// ---- DUTs/IO/Boxes/AT2042_33A3DF1B.TcDUT
{attribute 'GeneratedUsingTerminal: AT2042-5250-0019'}
{attribute addProperty BoxType "AT2042-5250-0019"}
{attribute addProperty Description "AT2042-5250 Sensor line with feed (B23-Connector), +45°"}
{attribute addProperty Physics "K"}
{attribute addProperty Id "FB_InputsAT %I*FB_Inputs_4BC4AA0166FB_OutputsAT %Q*FB_Outputs_DAFD38E02WcStateAT %I*WcState_9091E0EB2InfoDataAT %I*InfoData_A7436BC610"}
{attribute addProperty CRC "866377499"}
{attribute addProperty Size "80"}
TYPE AT2042_33A3DF1B EXTENDS EtcSlaveTerminalBase_947E5A46 :
STRUCT
	{attribute addProperty Name "FB_Inputs"}
	FB_Inputs : FB_Inputs_4BC4AA01;
	{attribute addProperty Name "FB_Outputs"}
	FB_Outputs : FB_Outputs_DAFD38E0;
	{attribute addProperty Name "WcState"}
	WcState : WcState_9091E0EB;
	{attribute addProperty Name "InfoData"}
	InfoData : InfoData_A7436BC6;
END_STRUCT
END_TYPE

// ---- DUTs/IO/Boxes/AT2041_33A3DF1B.TcDUT
{attribute 'GeneratedUsingTerminal: AT2041-5250-0019'}
{attribute addProperty BoxType "AT2041-5250-0019"}
{attribute addProperty Description "AT2041-5250 Sensor line with feed, +45°"}
{attribute addProperty Physics "K"}
{attribute addProperty Id "FB_InputsAT %I*FB_Inputs_4BC4AA0166FB_OutputsAT %Q*FB_Outputs_DAFD38E02WcStateAT %I*WcState_9091E0EB2InfoDataAT %I*InfoData_A7436BC610"}
{attribute addProperty CRC "866377499"}
{attribute addProperty Size "80"}
TYPE AT2041_33A3DF1B EXTENDS EtcSlaveTerminalBase_947E5A46 :
STRUCT
	{attribute addProperty Name "FB_Inputs"}
	FB_Inputs : FB_Inputs_4BC4AA01;
	{attribute addProperty Name "FB_Outputs"}
	FB_Outputs : FB_Outputs_DAFD38E0;
	{attribute addProperty Name "WcState"}
	WcState : WcState_9091E0EB;
	{attribute addProperty Name "InfoData"}
	InfoData : InfoData_A7436BC6;
END_STRUCT
END_TYPE

// ---- DUTs/IO/Boxes/AT2040_33A3DF1B.TcDUT
{attribute 'GeneratedUsingTerminal: AT2040-5250-0019'}
{attribute addProperty BoxType "AT2040-5250-0019"}
{attribute addProperty Description "AT2040-5250 Sensor line +45°"}
{attribute addProperty Physics "K"}
{attribute addProperty Id "FB_InputsAT %I*FB_Inputs_4BC4AA0166FB_OutputsAT %Q*FB_Outputs_DAFD38E02WcStateAT %I*WcState_9091E0EB2InfoDataAT %I*InfoData_A7436BC610"}
{attribute addProperty CRC "866377499"}
{attribute addProperty Size "80"}
TYPE AT2040_33A3DF1B EXTENDS EtcSlaveTerminalBase_947E5A46 :
STRUCT
	{attribute addProperty Name "FB_Inputs"}
	FB_Inputs : FB_Inputs_4BC4AA01;
	{attribute addProperty Name "FB_Outputs"}
	FB_Outputs : FB_Outputs_DAFD38E0;
	{attribute addProperty Name "WcState"}
	WcState : WcState_9091E0EB;
	{attribute addProperty Name "InfoData"}
	InfoData : InfoData_A7436BC6;
END_STRUCT
END_TYPE

// ---- DUTs/IO/Boxes/AT2042_2EA6C9BF.TcDUT
{attribute 'GeneratedUsingTerminal: AT2042-0250-0024'}
{attribute addProperty BoxType "AT2042-0250-0024"}
{attribute addProperty Description "AT2042-0250 Motor module with feed (B23-Connector), +45°, 250 mm, 48V"}
{attribute addProperty Physics "YKY"}
{attribute addProperty Id "CC_InputsAT %I*CC_Inputs_2C1C9EE032CC_OutputsAT %Q*CC_Outputs_69F9BE1432WcStateAT %I*WcState_9091E0EB2InfoDataAT %I*InfoData_BEF6B88E18"}
{attribute addProperty CRC "782682559"}
{attribute addProperty Size "84"}
TYPE AT2042_2EA6C9BF EXTENDS EtcSlaveBoxBase_77A0E4A7 :
STRUCT
	{attribute addProperty Name "CC_Inputs"}
	CC_Inputs : CC_Inputs_2C1C9EE0;
	{attribute addProperty Name "CC_Outputs"}
	CC_Outputs : CC_Outputs_69F9BE14;
	{attribute addProperty Name "WcState"}
	WcState : WcState_9091E0EB;
	{attribute addProperty Name "InfoData"}
	InfoData : InfoData_BEF6B88E;
END_STRUCT
END_TYPE

// ---- DUTs/IO/Boxes/AT2025_33A3DF1B.TcDUT
{attribute 'GeneratedUsingTerminal: AT2025-5250-0019'}
{attribute addProperty BoxType "AT2025-5250-0019"}
{attribute addProperty Description "AT2025-5250 Sensor line -22.5°"}
{attribute addProperty Physics "K"}
{attribute addProperty Id "FB_InputsAT %I*FB_Inputs_4BC4AA0166FB_OutputsAT %Q*FB_Outputs_DAFD38E02WcStateAT %I*WcState_9091E0EB2InfoDataAT %I*InfoData_A7436BC610"}
{attribute addProperty CRC "866377499"}
{attribute addProperty Size "80"}
TYPE AT2025_33A3DF1B EXTENDS EtcSlaveTerminalBase_947E5A46 :
STRUCT
	{attribute addProperty Name "FB_Inputs"}
	FB_Inputs : FB_Inputs_4BC4AA01;
	{attribute addProperty Name "FB_Outputs"}
	FB_Outputs : FB_Outputs_DAFD38E0;
	{attribute addProperty Name "WcState"}
	WcState : WcState_9091E0EB;
	{attribute addProperty Name "InfoData"}
	InfoData : InfoData_A7436BC6;
END_STRUCT
END_TYPE

// ---- DUTs/IO/Boxes/AT2050_2EA6C9BF.TcDUT
{attribute 'GeneratedUsingTerminal: AT2050-0500-0016'}
{attribute addProperty BoxType "AT2050-0500-0016"}
{attribute addProperty Description "AT2050-0500 Motor module, 90° clothoid, EtherCAT In, 50V"}
{attribute addProperty Physics "YKY"}
{attribute addProperty Id "CC_InputsAT %I*CC_Inputs_2C1C9EE032CC_OutputsAT %Q*CC_Outputs_69F9BE1432WcStateAT %I*WcState_9091E0EB2InfoDataAT %I*InfoData_BEF6B88E18"}
{attribute addProperty CRC "782682559"}
{attribute addProperty Size "84"}
TYPE AT2050_2EA6C9BF EXTENDS EtcSlaveBoxBase_77A0E4A7 :
STRUCT
	{attribute addProperty Name "CC_Inputs"}
	CC_Inputs : CC_Inputs_2C1C9EE0;
	{attribute addProperty Name "CC_Outputs"}
	CC_Outputs : CC_Outputs_69F9BE14;
	{attribute addProperty Name "WcState"}
	WcState : WcState_9091E0EB;
	{attribute addProperty Name "InfoData"}
	InfoData : InfoData_BEF6B88E;
END_STRUCT
END_TYPE

// ---- DUTs/IO/Boxes/AT2021_33A3DF1B.TcDUT
{attribute 'GeneratedUsingTerminal: AT2021-5250-0019'}
{attribute addProperty BoxType "AT2021-5250-0019"}
{attribute addProperty Description "AT2021-5250 Sensor line with feed, +22.5°"}
{attribute addProperty Physics "K"}
{attribute addProperty Id "FB_InputsAT %I*FB_Inputs_4BC4AA0166FB_OutputsAT %Q*FB_Outputs_DAFD38E02WcStateAT %I*WcState_9091E0EB2InfoDataAT %I*InfoData_A7436BC610"}
{attribute addProperty CRC "866377499"}
{attribute addProperty Size "80"}
TYPE AT2021_33A3DF1B EXTENDS EtcSlaveTerminalBase_947E5A46 :
STRUCT
	{attribute addProperty Name "FB_Inputs"}
	FB_Inputs : FB_Inputs_4BC4AA01;
	{attribute addProperty Name "FB_Outputs"}
	FB_Outputs : FB_Outputs_DAFD38E0;
	{attribute addProperty Name "WcState"}
	WcState : WcState_9091E0EB;
	{attribute addProperty Name "InfoData"}
	InfoData : InfoData_A7436BC6;
END_STRUCT
END_TYPE

// ---- DUTs/IO/Boxes/AT2020_33A3DF1B.TcDUT
{attribute 'GeneratedUsingTerminal: AT2020-5250-0019'}
{attribute addProperty BoxType "AT2020-5250-0019"}
{attribute addProperty Description "AT2020-5250 Sensor line +22.5°"}
{attribute addProperty Physics "K"}
{attribute addProperty Id "FB_InputsAT %I*FB_Inputs_4BC4AA0166FB_OutputsAT %Q*FB_Outputs_DAFD38E02WcStateAT %I*WcState_9091E0EB2InfoDataAT %I*InfoData_A7436BC610"}
{attribute addProperty CRC "866377499"}
{attribute addProperty Size "80"}
TYPE AT2020_33A3DF1B EXTENDS EtcSlaveTerminalBase_947E5A46 :
STRUCT
	{attribute addProperty Name "FB_Inputs"}
	FB_Inputs : FB_Inputs_4BC4AA01;
	{attribute addProperty Name "FB_Outputs"}
	FB_Outputs : FB_Outputs_DAFD38E0;
	{attribute addProperty Name "WcState"}
	WcState : WcState_9091E0EB;
	{attribute addProperty Name "InfoData"}
	InfoData : InfoData_A7436BC6;
END_STRUCT
END_TYPE

// ---- DUTs/IO/Boxes/AT2001_33A3DF1B.TcDUT
{attribute 'GeneratedUsingTerminal: AT2001-5250-0017'}
{attribute addProperty BoxType "AT2001-5250-0017"}
{attribute addProperty Description "AT2001-5250 Sensor line with feed"}
{attribute addProperty Physics "K"}
{attribute addProperty Id "FB_InputsAT %I*FB_Inputs_4BC4AA0166FB_OutputsAT %Q*FB_Outputs_DAFD38E02WcStateAT %I*WcState_9091E0EB2InfoDataAT %I*InfoData_A7436BC610"}
{attribute addProperty CRC "866377499"}
{attribute addProperty Size "80"}
TYPE AT2001_33A3DF1B EXTENDS EtcSlaveTerminalBase_947E5A46 :
STRUCT
	{attribute addProperty Name "FB_Inputs"}
	FB_Inputs : FB_Inputs_4BC4AA01;
	{attribute addProperty Name "FB_Outputs"}
	FB_Outputs : FB_Outputs_DAFD38E0;
	{attribute addProperty Name "WcState"}
	WcState : WcState_9091E0EB;
	{attribute addProperty Name "InfoData"}
	InfoData : InfoData_A7436BC6;
END_STRUCT
END_TYPE

// ---- DUTs/IO/Boxes/AT2002_33A3DF1B.TcDUT
{attribute 'GeneratedUsingTerminal: AT2002-5249-0018'}
{attribute addProperty BoxType "AT2002-5249-0018"}
{attribute addProperty Description "AT2002-5249 Sensor line (Track management) with feed"}
{attribute addProperty Physics "K"}
{attribute addProperty Id "FB_InputsAT %I*FB_Inputs_4BC4AA0166FB_OutputsAT %Q*FB_Outputs_DAFD38E02WcStateAT %I*WcState_9091E0EB2InfoDataAT %I*InfoData_A7436BC610"}
{attribute addProperty CRC "866377499"}
{attribute addProperty Size "80"}
TYPE AT2002_33A3DF1B EXTENDS EtcSlaveTerminalBase_947E5A46 :
STRUCT
	{attribute addProperty Name "FB_Inputs"}
	FB_Inputs : FB_Inputs_4BC4AA01;
	{attribute addProperty Name "FB_Outputs"}
	FB_Outputs : FB_Outputs_DAFD38E0;
	{attribute addProperty Name "WcState"}
	WcState : WcState_9091E0EB;
	{attribute addProperty Name "InfoData"}
	InfoData : InfoData_A7436BC6;
END_STRUCT
END_TYPE

// ---- DUTs/IO/Boxes/ATH2000_2EA6C9BF.TcDUT
{attribute 'GeneratedUsingTerminal: ATH2000-0250-0022'}
{attribute addProperty BoxType "ATH2000-0250-0022"}
{attribute addProperty Description "ATH2000-0250 Hygienic Motor module 250 mm, 48V"}
{attribute addProperty Physics "YKY"}
{attribute addProperty Id "CC_InputsAT %I*CC_Inputs_2C1C9EE032CC_OutputsAT %Q*CC_Outputs_69F9BE1432WcStateAT %I*WcState_9091E0EB2InfoDataAT %I*InfoData_BEF6B88E18"}
{attribute addProperty CRC "782682559"}
{attribute addProperty Size "84"}
TYPE ATH2000_2EA6C9BF EXTENDS EtcSlaveBoxBase_77A0E4A7 :
STRUCT
	{attribute addProperty Name "CC_Inputs"}
	CC_Inputs : CC_Inputs_2C1C9EE0;
	{attribute addProperty Name "CC_Outputs"}
	CC_Outputs : CC_Outputs_69F9BE14;
	{attribute addProperty Name "WcState"}
	WcState : WcState_9091E0EB;
	{attribute addProperty Name "InfoData"}
	InfoData : InfoData_BEF6B88E;
END_STRUCT
END_TYPE

// ---- DUTs/IO/Boxes/ATH2050_6EC099B7.TcDUT
{attribute 'GeneratedUsingTerminal: ATH2050-5501-0022'}
{attribute addProperty BoxType "ATH2050-5501-0022"}
{attribute addProperty Description "ATH2050-5501 Hygienic Sensor 90° clothoid, EtherCAT Out"}
{attribute addProperty Physics "K"}
{attribute addProperty Id "FB_InputsAT %I*FB_Inputs_391456510FB_OutputsAT %Q*FB_Outputs_DAFD38E02WcStateAT %I*WcState_9091E0EB2InfoDataAT %I*InfoData_A7436BC610"}
{attribute addProperty CRC "1858116023"}
{attribute addProperty Size "14"}
TYPE ATH2050_6EC099B7 EXTENDS EtcSlaveTerminalBase_947E5A46 :
STRUCT
	{attribute addProperty Name "FB_Inputs"}
	FB_Inputs : FB_Inputs_39145651;
	{attribute addProperty Name "FB_Outputs"}
	FB_Outputs : FB_Outputs_DAFD38E0;
	{attribute addProperty Name "WcState"}
	WcState : WcState_9091E0EB;
	{attribute addProperty Name "InfoData"}
	InfoData : InfoData_A7436BC6;
END_STRUCT
END_TYPE

// ---- DUTs/IO/Boxes/ATH2040_41437DDC.TcDUT
{attribute 'GeneratedUsingTerminal: ATH2040-5250-0022'}
{attribute addProperty BoxType "ATH2040-5250-0022"}
{attribute addProperty Description "ATH2040-5250 Hygienic Sensor +45°"}
{attribute addProperty Physics "K"}
{attribute addProperty Id "FB_InputsAT %I*FB_Inputs_01C600450FB_OutputsAT %Q*FB_Outputs_DAFD38E02WcStateAT %I*WcState_9091E0EB2InfoDataAT %I*InfoData_A7436BC610"}
{attribute addProperty CRC "1094942172"}
{attribute addProperty Size "14"}
TYPE ATH2040_41437DDC EXTENDS EtcSlaveTerminalBase_947E5A46 :
STRUCT
	{attribute addProperty Name "FB_Inputs"}
	FB_Inputs : FB_Inputs_01C60045;
	{attribute addProperty Name "FB_Outputs"}
	FB_Outputs : FB_Outputs_DAFD38E0;
	{attribute addProperty Name "WcState"}
	WcState : WcState_9091E0EB;
	{attribute addProperty Name "InfoData"}
	InfoData : InfoData_A7436BC6;
END_STRUCT
END_TYPE

// ---- DUTs/IO/Boxes/ATH2040_2EA6C9BF.TcDUT
{attribute 'GeneratedUsingTerminal: ATH2040-0250-0022'}
{attribute addProperty BoxType "ATH2040-0250-0022"}
{attribute addProperty Description "ATH2040-0250 Hygienic Motor module +45°, 250mm, 48V"}
{attribute addProperty Physics "YKY"}
{attribute addProperty Id "CC_InputsAT %I*CC_Inputs_2C1C9EE032CC_OutputsAT %Q*CC_Outputs_69F9BE1432WcStateAT %I*WcState_9091E0EB2InfoDataAT %I*InfoData_BEF6B88E18"}
{attribute addProperty CRC "782682559"}
{attribute addProperty Size "84"}
TYPE ATH2040_2EA6C9BF EXTENDS EtcSlaveBoxBase_77A0E4A7 :
STRUCT
	{attribute addProperty Name "CC_Inputs"}
	CC_Inputs : CC_Inputs_2C1C9EE0;
	{attribute addProperty Name "CC_Outputs"}
	CC_Outputs : CC_Outputs_69F9BE14;
	{attribute addProperty Name "WcState"}
	WcState : WcState_9091E0EB;
	{attribute addProperty Name "InfoData"}
	InfoData : InfoData_BEF6B88E;
END_STRUCT
END_TYPE

// ---- DUTs/IO/Boxes/ATH2050_2EA6C9BF.TcDUT
{attribute 'GeneratedUsingTerminal: ATH2050-0500-0022'}
{attribute addProperty BoxType "ATH2050-0500-0022"}
{attribute addProperty Description "ATH2050-0500 Hygienic Motor module 90° clothoid, EtherCAT In"}
{attribute addProperty Physics "YKY"}
{attribute addProperty Id "CC_InputsAT %I*CC_Inputs_2C1C9EE032CC_OutputsAT %Q*CC_Outputs_69F9BE1432WcStateAT %I*WcState_9091E0EB2InfoDataAT %I*InfoData_BEF6B88E18"}
{attribute addProperty CRC "782682559"}
{attribute addProperty Size "84"}
TYPE ATH2050_2EA6C9BF EXTENDS EtcSlaveBoxBase_77A0E4A7 :
STRUCT
	{attribute addProperty Name "CC_Inputs"}
	CC_Inputs : CC_Inputs_2C1C9EE0;
	{attribute addProperty Name "CC_Outputs"}
	CC_Outputs : CC_Outputs_69F9BE14;
	{attribute addProperty Name "WcState"}
	WcState : WcState_9091E0EB;
	{attribute addProperty Name "InfoData"}
	InfoData : InfoData_BEF6B88E;
END_STRUCT
END_TYPE

// ---- DUTs/IO/Boxes/ATH2000_D874080E.TcDUT
{attribute 'GeneratedUsingTerminal: ATH2000-5250-0022'}
{attribute addProperty BoxType "ATH2000-5250-0022"}
{attribute addProperty Description "ATH2000-5250 Hygienic Sensor line"}
{attribute addProperty Physics "K"}
{attribute addProperty Id "FB_InputsAT %I*FB_Inputs_2D6658510FB_OutputsAT %Q*FB_Outputs_DAFD38E02WcStateAT %I*WcState_9091E0EB2InfoDataAT %I*InfoData_A7436BC610"}
{attribute addProperty CRC "3631482894"}
{attribute addProperty Size "14"}
TYPE ATH2000_D874080E EXTENDS EtcSlaveTerminalBase_947E5A46 :
STRUCT
	{attribute addProperty Name "FB_Inputs"}
	FB_Inputs : FB_Inputs_2D665851;
	{attribute addProperty Name "FB_Outputs"}
	FB_Outputs : FB_Outputs_DAFD38E0;
	{attribute addProperty Name "WcState"}
	WcState : WcState_9091E0EB;
	{attribute addProperty Name "InfoData"}
	InfoData : InfoData_A7436BC6;
END_STRUCT
END_TYPE

// ---- DUTs/IO/Devices/SyncUnitTask_2D604ED5.TcDUT
{attribute 'GeneratedUsingTerminal: IODEVICETYPE_ETHERCATPROT'}
{attribute addProperty BoxType "IODEVICETYPE_ETHERCATPROT"}
{attribute addProperty Id "WcStateAT %I*WcState_0B2B16F91InfoDataAT %I*InfoData_2A97D6CF8"}
{attribute addProperty CRC "761286357"}
{attribute addProperty Size "9"}
TYPE SyncUnitTask_2D604ED5 :
STRUCT
	{attribute addProperty Name "WcState"}
	WcState : WcState_0B2B16F9;
	{attribute addProperty Name "InfoData"}
	InfoData : InfoData_2A97D6CF;
END_STRUCT
END_TYPE

// ---- DUTs/IO/Devices/SyncUnitTasks_6FEB8257.TcDUT
{attribute 'GeneratedUsingTerminal: '}
{attribute addProperty BoxType ""}
{attribute addProperty Id "unreferencedAT %I*SyncUnitTask_2D604ED59PlcTaskAT %I*SyncUnitTask_2D604ED59"}
{attribute addProperty CRC "1877705303"}
{attribute addProperty Size "18"}
TYPE SyncUnitTasks_6FEB8257 :
STRUCT
	{attribute addProperty Name "unreferenced"}
	unreferenced : SyncUnitTask_2D604ED5;
	{attribute addProperty Name "PlcTask"}
	PlcTask : SyncUnitTask_2D604ED5;
END_STRUCT
END_TYPE

// ---- DUTs/IO/Devices/SyncUnits_99E584AF.TcDUT
{attribute 'GeneratedUsingTerminal: '}
{attribute addProperty BoxType ""}
{attribute addProperty Id "_defaultAT %I*SyncUnitTasks_6FEB825718"}
{attribute addProperty CRC "2581955759"}
{attribute addProperty Size "18"}
TYPE SyncUnits_99E584AF :
STRUCT
	{attribute addProperty Name "_default"}
	_default : SyncUnitTasks_6FEB8257;
END_STRUCT
END_TYPE

// ---- DUTs/IO/Topology/A_0060_AT2020_0250_0019_AT2020_0250_29EE8276.TcDUT
{attribute 'GeneratedUsingTerminal: AT2020-0250-0019'}
{attribute addProperty BoxType "AT2020-0250-0019"}
{attribute addProperty Id "A_0085_AT2050_5500_0018_AT2050_5500AT2050_33A3DF1B80"}
{attribute addProperty CRC "703496822"}
{attribute addProperty Size "80"}
{attribute addProperty Name "A_0060(AT2020-0250-0019) (AT2020-0250)"}
TYPE A_0060_AT2020_0250_0019_AT2020_0250_29EE8276 EXTENDS AT2020_2EA6C9BF :
STRUCT
	{attribute addProperty Name "A_0085(AT2050-5500-0018) (AT2050-5500)"}
	{attribute addProperty PreviousPort "A_0060(AT2020-0250-0019) (AT2020-0250) : B"}
	A_0085_AT2050_5500_0018_AT2050_5500 : AT2050_33A3DF1B;
END_STRUCT
END_TYPE

// ---- DUTs/IO/Topology/A_0036_AT2040_0250_0021_0B822AE4.TcDUT
{attribute 'GeneratedUsingTerminal: AT2040-0250-0021'}
{attribute addProperty BoxType "AT2040-0250-0021"}
{attribute addProperty Id "A_0108_AT2000_5233_0019_AT2000_5233AT2000_33A3DF1B80"}
{attribute addProperty CRC "193080036"}
{attribute addProperty Size "80"}
{attribute addProperty Name "A_0036(AT2040-0250-0021)"}
TYPE A_0036_AT2040_0250_0021_0B822AE4 EXTENDS AT2040_2EA6C9BF :
STRUCT
	{attribute addProperty Name "A_0108(AT2000-5233-0019) (AT2000-5233)"}
	{attribute addProperty PreviousPort "A_0036(AT2040-0250-0021) : B"}
	A_0108_AT2000_5233_0019_AT2000_5233 : AT2000_33A3DF1B;
END_STRUCT
END_TYPE

// ---- DUTs/IO/Topology/A_0037_AT2040_0250_0022_033DCEC4.TcDUT
{attribute 'GeneratedUsingTerminal: AT2040-0250-0022'}
{attribute addProperty BoxType "AT2040-0250-0022"}
{attribute addProperty Id "A_0107_AT2000_5233_0018_AT2000_5233AT2000_33A3DF1B80"}
{attribute addProperty CRC "54382276"}
{attribute addProperty Size "80"}
{attribute addProperty Name "A_0037(AT2040-0250-0022)"}
TYPE A_0037_AT2040_0250_0022_033DCEC4 EXTENDS AT2040_2EA6C9BF :
STRUCT
	{attribute addProperty Name "A_0107(AT2000-5233-0018) (AT2000-5233)"}
	{attribute addProperty PreviousPort "A_0037(AT2040-0250-0022) : B"}
	A_0107_AT2000_5233_0018_AT2000_5233 : AT2000_33A3DF1B;
END_STRUCT
END_TYPE

// ---- DUTs/IO/Topology/A_0038_AT2040_0250_0023_C339CA0C.TcDUT
{attribute 'GeneratedUsingTerminal: AT2040-0250-0023'}
{attribute addProperty BoxType "AT2040-0250-0023"}
{attribute addProperty Id "A_0106_AT2026_5250_0019_AT2026_5250AT2026_33A3DF1B80"}
{attribute addProperty CRC "3275344396"}
{attribute addProperty Size "80"}
{attribute addProperty Name "A_0038(AT2040-0250-0023)"}
TYPE A_0038_AT2040_0250_0023_C339CA0C EXTENDS AT2040_2EA6C9BF :
STRUCT
	{attribute addProperty Name "A_0106(AT2026-5250-0019) (AT2026-5250)"}
	{attribute addProperty PreviousPort "A_0038(AT2040-0250-0023) : B"}
	A_0106_AT2026_5250_0019_AT2026_5250 : AT2026_33A3DF1B;
END_STRUCT
END_TYPE

// ---- DUTs/IO/Topology/A_0039_AT2040_0250_0024_375958EA.TcDUT
{attribute 'GeneratedUsingTerminal: AT2040-0250-0024'}
{attribute addProperty BoxType "AT2040-0250-0024"}
{attribute addProperty Id "A_0105_AT2026_5250_0018_AT2026_5250AT2026_33A3DF1B80"}
{attribute addProperty CRC "928602346"}
{attribute addProperty Size "80"}
{attribute addProperty Name "A_0039(AT2040-0250-0024)"}
TYPE A_0039_AT2040_0250_0024_375958EA EXTENDS AT2040_2EA6C9BF :
STRUCT
	{attribute addProperty Name "A_0105(AT2026-5250-0018) (AT2026-5250)"}
	{attribute addProperty PreviousPort "A_0039(AT2040-0250-0024) : B"}
	A_0105_AT2026_5250_0018_AT2026_5250 : AT2026_33A3DF1B;
END_STRUCT
END_TYPE

// ---- DUTs/IO/Topology/A_0040_AT2041_0250_0018_536500F2.TcDUT
{attribute 'GeneratedUsingTerminal: AT2041-0250-0018'}
{attribute addProperty BoxType "AT2041-0250-0018"}
{attribute addProperty Id "A_0104_AT2042_5250_0019_AT2042_5250AT2042_33A3DF1B80"}
{attribute addProperty CRC "1399128306"}
{attribute addProperty Size "80"}
{attribute addProperty Name "A_0040(AT2041-0250-0018)"}
TYPE A_0040_AT2041_0250_0018_536500F2 EXTENDS AT2041_2EA6C9BF :
STRUCT
	{attribute addProperty Name "A_0104(AT2042-5250-0019) (AT2042-5250)"}
	{attribute addProperty PreviousPort "A_0040(AT2041-0250-0018) : B"}
	A_0104_AT2042_5250_0019_AT2042_5250 : AT2042_33A3DF1B;
END_STRUCT
END_TYPE

// ---- DUTs/IO/Topology/A_0041_AT2041_0250_0019_F34F4056.TcDUT
{attribute 'GeneratedUsingTerminal: AT2041-0250-0019'}
{attribute addProperty BoxType "AT2041-0250-0019"}
{attribute addProperty Id "A_0103_AT2042_5250_0018_AT2042_5250AT2042_33A3DF1B80"}
{attribute addProperty CRC "4082057302"}
{attribute addProperty Size "80"}
{attribute addProperty Name "A_0041(AT2041-0250-0019)"}
TYPE A_0041_AT2041_0250_0019_F34F4056 EXTENDS AT2041_2EA6C9BF :
STRUCT
	{attribute addProperty Name "A_0103(AT2042-5250-0018) (AT2042-5250)"}
	{attribute addProperty PreviousPort "A_0041(AT2041-0250-0019) : B"}
	A_0103_AT2042_5250_0018_AT2042_5250 : AT2042_33A3DF1B;
END_STRUCT
END_TYPE

// ---- DUTs/IO/Topology/A_0042_AT2041_0250_0020_5E65A51E.TcDUT
{attribute 'GeneratedUsingTerminal: AT2041-0250-0020'}
{attribute addProperty BoxType "AT2041-0250-0020"}
{attribute addProperty Id "A_0102_AT2041_5250_0019_AT2041_5250AT2041_33A3DF1B80"}
{attribute addProperty CRC "1583719710"}
{attribute addProperty Size "80"}
{attribute addProperty Name "A_0042(AT2041-0250-0020)"}
TYPE A_0042_AT2041_0250_0020_5E65A51E EXTENDS AT2041_2EA6C9BF :
STRUCT
	{attribute addProperty Name "A_0102(AT2041-5250-0019) (AT2041-5250)"}
	{attribute addProperty PreviousPort "A_0042(AT2041-0250-0020) : B"}
	A_0102_AT2041_5250_0019_AT2041_5250 : AT2041_33A3DF1B;
END_STRUCT
END_TYPE

// ---- DUTs/IO/Topology/A_0043_AT2041_0250_0021_AA0537F8.TcDUT
{attribute 'GeneratedUsingTerminal: AT2041-0250-0021'}
{attribute addProperty BoxType "AT2041-0250-0021"}
{attribute addProperty Id "A_0101_AT2041_5250_0018_AT2041_5250AT2041_33A3DF1B80"}
{attribute addProperty CRC "2852468728"}
{attribute addProperty Size "80"}
{attribute addProperty Name "A_0043(AT2041-0250-0021)"}
TYPE A_0043_AT2041_0250_0021_AA0537F8 EXTENDS AT2041_2EA6C9BF :
STRUCT
	{attribute addProperty Name "A_0101(AT2041-5250-0018) (AT2041-5250)"}
	{attribute addProperty PreviousPort "A_0043(AT2041-0250-0021) : B"}
	A_0101_AT2041_5250_0018_AT2041_5250 : AT2041_33A3DF1B;
END_STRUCT
END_TYPE

// ---- DUTs/IO/Topology/A_0044_AT2041_0250_0022_5A9A39BA.TcDUT
{attribute 'GeneratedUsingTerminal: AT2041-0250-0022'}
{attribute addProperty BoxType "AT2041-0250-0022"}
{attribute addProperty Id "A_0100_AT2040_5250_0019_AT2040_5250AT2040_33A3DF1B80"}
{attribute addProperty CRC "1520056762"}
{attribute addProperty Size "80"}
{attribute addProperty Name "A_0044(AT2041-0250-0022)"}
TYPE A_0044_AT2041_0250_0022_5A9A39BA EXTENDS AT2041_2EA6C9BF :
STRUCT
	{attribute addProperty Name "A_0100(AT2040-5250-0019) (AT2040-5250)"}
	{attribute addProperty PreviousPort "A_0044(AT2041-0250-0022) : B"}
	A_0100_AT2040_5250_0019_AT2040_5250 : AT2040_33A3DF1B;
END_STRUCT
END_TYPE

// ---- DUTs/IO/Topology/A_0045_AT2041_0250_0023_51C662AC.TcDUT
{attribute 'GeneratedUsingTerminal: AT2041-0250-0023'}
{attribute addProperty BoxType "AT2041-0250-0023"}
{attribute addProperty Id "A_0099_AT2040_5250_0018_AT2040_5250AT2040_33A3DF1B80"}
{attribute addProperty CRC "1371955884"}
{attribute addProperty Size "80"}
{attribute addProperty Name "A_0045(AT2041-0250-0023)"}
TYPE A_0045_AT2041_0250_0023_51C662AC EXTENDS AT2041_2EA6C9BF :
STRUCT
	{attribute addProperty Name "A_0099(AT2040-5250-0018) (AT2040-5250)"}
	{attribute addProperty PreviousPort "A_0045(AT2041-0250-0023) : B"}
	A_0099_AT2040_5250_0018_AT2040_5250 : AT2040_33A3DF1B;
END_STRUCT
END_TYPE

// ---- DUTs/IO/Topology/A_0046_AT2042_0250_0024_1B20CF31.TcDUT
{attribute 'GeneratedUsingTerminal: AT2042-0250-0024'}
{attribute addProperty BoxType "AT2042-0250-0024"}
{attribute addProperty Id "A_0098_AT2025_5250_0019_AT2025_5250AT2025_33A3DF1B80"}
{attribute addProperty CRC "455135025"}
{attribute addProperty Size "80"}
{attribute addProperty Name "A_0046(AT2042-0250-0024)"}
TYPE A_0046_AT2042_0250_0024_1B20CF31 EXTENDS AT2042_2EA6C9BF :
STRUCT
	{attribute addProperty Name "A_0098(AT2025-5250-0019) (AT2025-5250)"}
	{attribute addProperty PreviousPort "A_0046(AT2042-0250-0024) : B"}
	A_0098_AT2025_5250_0019_AT2025_5250 : AT2025_33A3DF1B;
END_STRUCT
END_TYPE

// ---- DUTs/IO/Topology/A_0047_AT2050_0500_0016_139F2B11.TcDUT
{attribute 'GeneratedUsingTerminal: AT2050-0500-0016'}
{attribute addProperty BoxType "AT2050-0500-0016"}
{attribute addProperty Id "A_0097_AT2025_5250_0018_AT2025_5250AT2025_33A3DF1B80"}
{attribute addProperty CRC "329198353"}
{attribute addProperty Size "80"}
{attribute addProperty Name "A_0047(AT2050-0500-0016)"}
TYPE A_0047_AT2050_0500_0016_139F2B11 EXTENDS AT2050_2EA6C9BF :
STRUCT
	{attribute addProperty Name "A_0097(AT2025-5250-0018) (AT2025-5250)"}
	{attribute addProperty PreviousPort "A_0047(AT2050-0500-0016) : B"}
	A_0097_AT2025_5250_0018_AT2025_5250 : AT2025_33A3DF1B;
END_STRUCT
END_TYPE

// ---- DUTs/IO/Topology/A_0048_AT2050_0500_0017_3F977F47.TcDUT
{attribute 'GeneratedUsingTerminal: AT2050-0500-0017'}
{attribute addProperty BoxType "AT2050-0500-0017"}
{attribute addProperty Id "A_0096_AT2025_5250_0017_AT2025_5250AT2025_33A3DF1B80"}
{attribute addProperty CRC "1066893127"}
{attribute addProperty Size "80"}
{attribute addProperty Name "A_0048(AT2050-0500-0017)"}
TYPE A_0048_AT2050_0500_0017_3F977F47 EXTENDS AT2050_2EA6C9BF :
STRUCT
	{attribute addProperty Name "A_0096(AT2025-5250-0017) (AT2025-5250)"}
	{attribute addProperty PreviousPort "A_0048(AT2050-0500-0017) : B"}
	A_0096_AT2025_5250_0017_AT2025_5250 : AT2025_33A3DF1B;
END_STRUCT
END_TYPE

// ---- DUTs/IO/Topology/A_0049_AT2050_0500_0018_CBE655A8.TcDUT
{attribute 'GeneratedUsingTerminal: AT2050-0500-0018'}
{attribute addProperty BoxType "AT2050-0500-0018"}
{attribute addProperty Id "A_0095_AT2021_5250_0019_AT2021_5250AT2021_33A3DF1B80"}
{attribute addProperty CRC "3420870056"}
{attribute addProperty Size "80"}
{attribute addProperty Name "A_0049(AT2050-0500-0018)"}
TYPE A_0049_AT2050_0500_0018_CBE655A8 EXTENDS AT2050_2EA6C9BF :
STRUCT
	{attribute addProperty Name "A_0095(AT2021-5250-0019) (AT2021-5250)"}
	{attribute addProperty PreviousPort "A_0049(AT2050-0500-0018) : B"}
	A_0095_AT2021_5250_0019_AT2021_5250 : AT2021_33A3DF1B;
END_STRUCT
END_TYPE

// ---- DUTs/IO/Topology/A_0050_AT2050_0500_0019_15A3AE6F.TcDUT
{attribute 'GeneratedUsingTerminal: AT2050-0500-0019'}
{attribute addProperty BoxType "AT2050-0500-0019"}
{attribute addProperty Id "A_0094_AT2021_5250_0018_AT2021_5250AT2021_33A3DF1B80"}
{attribute addProperty CRC "363048559"}
{attribute addProperty Size "80"}
{attribute addProperty Name "A_0050(AT2050-0500-0019)"}
TYPE A_0050_AT2050_0500_0019_15A3AE6F EXTENDS AT2050_2EA6C9BF :
STRUCT
	{attribute addProperty Name "A_0094(AT2021-5250-0018) (AT2021-5250)"}
	{attribute addProperty PreviousPort "A_0050(AT2050-0500-0019) : B"}
	A_0094_AT2021_5250_0018_AT2021_5250 : AT2021_33A3DF1B;
END_STRUCT
END_TYPE

// ---- DUTs/IO/Topology/A_0051_AT2050_0500_0020_9B531B4E.TcDUT
{attribute 'GeneratedUsingTerminal: AT2050-0500-0020'}
{attribute addProperty BoxType "AT2050-0500-0020"}
{attribute addProperty Id "A_0093_AT2020_5250_0019_AT2020_5250AT2020_33A3DF1B80"}
{attribute addProperty CRC "2605914958"}
{attribute addProperty Size "80"}
{attribute addProperty Name "A_0051(AT2050-0500-0020)"}
TYPE A_0051_AT2050_0500_0020_9B531B4E EXTENDS AT2050_2EA6C9BF :
STRUCT
	{attribute addProperty Name "A_0093(AT2020-5250-0019) (AT2020-5250)"}
	{attribute addProperty PreviousPort "A_0051(AT2050-0500-0020) : B"}
	A_0093_AT2020_5250_0019_AT2020_5250 : AT2020_33A3DF1B;
END_STRUCT
END_TYPE

// ---- DUTs/IO/Topology/A_0052_AT2050_0500_0021_4516E089.TcDUT
{attribute 'GeneratedUsingTerminal: AT2050-0500-0021'}
{attribute addProperty BoxType "AT2050-0500-0021"}
{attribute addProperty Id "A_0092_AT2020_5250_0018_AT2020_5250AT2020_33A3DF1B80"}
{attribute addProperty CRC "1159127177"}
{attribute addProperty Size "80"}
{attribute addProperty Name "A_0052(AT2050-0500-0021)"}
TYPE A_0052_AT2050_0500_0021_4516E089 EXTENDS AT2050_2EA6C9BF :
STRUCT
	{attribute addProperty Name "A_0092(AT2020-5250-0018) (AT2020-5250)"}
	{attribute addProperty PreviousPort "A_0052(AT2050-0500-0021) : B"}
	A_0092_AT2020_5250_0018_AT2020_5250 : AT2020_33A3DF1B;
END_STRUCT
END_TYPE

// ---- DUTs/IO/Topology/A_0053_AT2050_0500_0022_433BDDFE.TcDUT
{attribute 'GeneratedUsingTerminal: AT2050-0500-0022'}
{attribute addProperty BoxType "AT2050-0500-0022"}
{attribute addProperty Id "A_0091_AT2020_5250_0017_AT2020_5250AT2020_33A3DF1B80"}
{attribute addProperty CRC "1127996926"}
{attribute addProperty Size "80"}
{attribute addProperty Name "A_0053(AT2050-0500-0022)"}
TYPE A_0053_AT2050_0500_0022_433BDDFE EXTENDS AT2050_2EA6C9BF :
STRUCT
	{attribute addProperty Name "A_0091(AT2020-5250-0017) (AT2020-5250)"}
	{attribute addProperty PreviousPort "A_0053(AT2050-0500-0022) : B"}
	A_0091_AT2020_5250_0017_AT2020_5250 : AT2020_33A3DF1B;
END_STRUCT
END_TYPE

// ---- DUTs/IO/Topology/A_0054_AT2050_0500_0023_B2F2DF55.TcDUT
{attribute 'GeneratedUsingTerminal: AT2050-0500-0023'}
{attribute addProperty BoxType "AT2050-0500-0023"}
{attribute addProperty Id "A_0090_AT2050_5501_0019_AT2050_5501AT2050_33A3DF1B80"}
{attribute addProperty CRC "3002261333"}
{attribute addProperty Size "80"}
{attribute addProperty Name "A_0054(AT2050-0500-0023)"}
TYPE A_0054_AT2050_0500_0023_B2F2DF55 EXTENDS AT2050_2EA6C9BF :
STRUCT
	{attribute addProperty Name "A_0090(AT2050-5501-0019) (AT2050-5501)"}
	{attribute addProperty PreviousPort "A_0054(AT2050-0500-0023) : B"}
	A_0090_AT2050_5501_0019_AT2050_5501 : AT2050_33A3DF1B;
END_STRUCT
END_TYPE

// ---- DUTs/IO/Topology/A_0055_AT2050_0500_0024_8D42A08D.TcDUT
{attribute 'GeneratedUsingTerminal: AT2050-0500-0024'}
{attribute addProperty BoxType "AT2050-0500-0024"}
{attribute addProperty Id "A_0089_AT2050_5501_0018_AT2050_5501AT2050_33A3DF1B80"}
{attribute addProperty CRC "2369953933"}
{attribute addProperty Size "80"}
{attribute addProperty Name "A_0055(AT2050-0500-0024)"}
TYPE A_0055_AT2050_0500_0024_8D42A08D EXTENDS AT2050_2EA6C9BF :
STRUCT
	{attribute addProperty Name "A_0089(AT2050-5501-0018) (AT2050-5501)"}
	{attribute addProperty PreviousPort "A_0055(AT2050-0500-0024) : B"}
	A_0089_AT2050_5501_0018_AT2050_5501 : AT2050_33A3DF1B;
END_STRUCT
END_TYPE

// ---- DUTs/IO/Topology/A_0056_AT2050_0501_0017_A14AF4DB.TcDUT
{attribute 'GeneratedUsingTerminal: AT2050-0501-0017'}
{attribute addProperty BoxType "AT2050-0501-0017"}
{attribute addProperty Id "A_0088_AT2050_5501_0017_AT2050_5501AT2050_33A3DF1B80"}
{attribute addProperty CRC "2706044123"}
{attribute addProperty Size "80"}
{attribute addProperty Name "A_0056(AT2050-0501-0017)"}
TYPE A_0056_AT2050_0501_0017_A14AF4DB EXTENDS AT2050_2EA6C9BF :
STRUCT
	{attribute addProperty Name "A_0088(AT2050-5501-0017) (AT2050-5501)"}
	{attribute addProperty PreviousPort "A_0056(AT2050-0501-0017) : B"}
	A_0088_AT2050_5501_0017_AT2050_5501 : AT2050_33A3DF1B;
END_STRUCT
END_TYPE

// ---- DUTs/IO/Topology/A_0057_AT2050_0501_0020_A9F510FB.TcDUT
{attribute 'GeneratedUsingTerminal: AT2050-0501-0020'}
{attribute addProperty BoxType "AT2050-0501-0020"}
{attribute addProperty Id "A_0087_AT2050_5501_0016_AT2050_5501AT2050_33A3DF1B80"}
{attribute addProperty CRC "2851410171"}
{attribute addProperty Size "80"}
{attribute addProperty Name "A_0057(AT2050-0501-0020)"}
TYPE A_0057_AT2050_0501_0020_A9F510FB EXTENDS AT2050_2EA6C9BF :
STRUCT
	{attribute addProperty Name "A_0087(AT2050-5501-0016) (AT2050-5501)"}
	{attribute addProperty PreviousPort "A_0057(AT2050-0501-0020) : B"}
	A_0087_AT2050_5501_0016_AT2050_5501 : AT2050_33A3DF1B;
END_STRUCT
END_TYPE

// ---- DUTs/IO/Topology/A_0058_AT2050_0501_0021_DD8E1090.TcDUT
{attribute 'GeneratedUsingTerminal: AT2050-0501-0021'}
{attribute addProperty BoxType "AT2050-0501-0021"}
{attribute addProperty Id "A_0086_AT2050_5500_0019_AT2050_5500AT2050_33A3DF1B80"}
{attribute addProperty CRC "3717075088"}
{attribute addProperty Size "80"}
{attribute addProperty Name "A_0058(AT2050-0501-0021)"}
TYPE A_0058_AT2050_0501_0021_DD8E1090 EXTENDS AT2050_2EA6C9BF :
STRUCT
	{attribute addProperty Name "A_0086(AT2050-5500-0019) (AT2050-5500)"}
	{attribute addProperty PreviousPort "A_0058(AT2050-0501-0021) : B"}
	A_0086_AT2050_5500_0019_AT2050_5500 : AT2050_33A3DF1B;
END_STRUCT
END_TYPE

// ---- DUTs/IO/Topology/A_0061_AT2020_0250_0023_AT2020_0250_2D9AB3DC.TcDUT
{attribute 'GeneratedUsingTerminal: AT2020-0250-0023'}
{attribute addProperty BoxType "AT2020-0250-0023"}
{attribute addProperty Id "A_0073_AT2000_5250_0016_AT2000_5250AT2000_33A3DF1B80"}
{attribute addProperty CRC "765113308"}
{attribute addProperty Size "80"}
{attribute addProperty Name "A_0061(AT2020-0250-0023) (AT2020-0250)"}
TYPE A_0061_AT2020_0250_0023_AT2020_0250_2D9AB3DC EXTENDS AT2020_2EA6C9BF :
STRUCT
	{attribute addProperty Name "A_0073(AT2000-5250-0016) (AT2000-5250)"}
	{attribute addProperty PreviousPort "A_0061(AT2020-0250-0023) (AT2020-0250) : B"}
	A_0073_AT2000_5250_0016_AT2000_5250 : AT2000_33A3DF1B;
END_STRUCT
END_TYPE

// ---- DUTs/IO/Topology/A_0062_AT2025_0250_0020_AT2025_0250_8DB0F378.TcDUT
{attribute 'GeneratedUsingTerminal: AT2025-0250-0020'}
{attribute addProperty BoxType "AT2025-0250-0020"}
{attribute addProperty Id "A_0074_AT2000_5250_0017_AT2000_5250AT2000_33A3DF1B80"}
{attribute addProperty CRC "2377184120"}
{attribute addProperty Size "80"}
{attribute addProperty Name "A_0062(AT2025-0250-0020) (AT2025-0250)"}
TYPE A_0062_AT2025_0250_0020_AT2025_0250_8DB0F378 EXTENDS AT2025_2EA6C9BF :
STRUCT
	{attribute addProperty Name "A_0074(AT2000-5250-0017) (AT2000-5250)"}
	{attribute addProperty PreviousPort "A_0062(AT2025-0250-0020) (AT2025-0250) : B"}
	A_0074_AT2000_5250_0017_AT2000_5250 : AT2000_33A3DF1B;
END_STRUCT
END_TYPE

// ---- DUTs/IO/Topology/A_0063_AT2025_0250_0022_AT2025_0250_E88F66A2.TcDUT
{attribute 'GeneratedUsingTerminal: AT2025-0250-0022'}
{attribute addProperty BoxType "AT2025-0250-0022"}
{attribute addProperty Id "A_0075_AT2000_5250_0019_AT2000_5250AT2000_33A3DF1B80"}
{attribute addProperty CRC "3901712034"}
{attribute addProperty Size "80"}
{attribute addProperty Name "A_0063(AT2025-0250-0022) (AT2025-0250)"}
TYPE A_0063_AT2025_0250_0022_AT2025_0250_E88F66A2 EXTENDS AT2025_2EA6C9BF :
STRUCT
	{attribute addProperty Name "A_0075(AT2000-5250-0019) (AT2000-5250)"}
	{attribute addProperty PreviousPort "A_0063(AT2025-0250-0022) (AT2025-0250) : B"}
	A_0075_AT2000_5250_0019_AT2000_5250 : AT2000_33A3DF1B;
END_STRUCT
END_TYPE

// ---- DUTs/IO/Topology/A_0064_AT2025_0250_0023_AT2025_0250_894F6FDC.TcDUT
{attribute 'GeneratedUsingTerminal: AT2025-0250-0023'}
{attribute addProperty BoxType "AT2025-0250-0023"}
{attribute addProperty Id "A_0076_AT2001_5250_0017_AT2001_5250AT2001_33A3DF1B80"}
{attribute addProperty CRC "2303684572"}
{attribute addProperty Size "80"}
{attribute addProperty Name "A_0064(AT2025-0250-0023) (AT2025-0250)"}
TYPE A_0064_AT2025_0250_0023_AT2025_0250_894F6FDC EXTENDS AT2025_2EA6C9BF :
STRUCT
	{attribute addProperty Name "A_0076(AT2001-5250-0017) (AT2001-5250)"}
	{attribute addProperty PreviousPort "A_0064(AT2025-0250-0023) (AT2025-0250) : B"}
	A_0076_AT2001_5250_0017_AT2001_5250 : AT2001_33A3DF1B;
END_STRUCT
END_TYPE

// ---- DUTs/IO/Topology/A_0065_AT2026_0250_0019_AT2026_0250_A5473B8A.TcDUT
{attribute 'GeneratedUsingTerminal: AT2026-0250-0019'}
{attribute addProperty BoxType "AT2026-0250-0019"}
{attribute addProperty Id "A_0077_AT2001_5250_0018_AT2001_5250AT2001_33A3DF1B80"}
{attribute addProperty CRC "2772908938"}
{attribute addProperty Size "80"}
{attribute addProperty Name "A_0065(AT2026-0250-0019) (AT2026-0250)"}
TYPE A_0065_AT2026_0250_0019_AT2026_0250_A5473B8A EXTENDS AT2026_2EA6C9BF :
STRUCT
	{attribute addProperty Name "A_0077(AT2001-5250-0018) (AT2001-5250)"}
	{attribute addProperty PreviousPort "A_0065(AT2026-0250-0019) (AT2026-0250) : B"}
	A_0077_AT2001_5250_0018_AT2001_5250 : AT2001_33A3DF1B;
END_STRUCT
END_TYPE

// ---- DUTs/IO/Topology/A_0066_AT2026_0250_0020_AT2026_0250_ADF8DFAA.TcDUT
{attribute 'GeneratedUsingTerminal: AT2026-0250-0020'}
{attribute addProperty BoxType "AT2026-0250-0020"}
{attribute addProperty Id "A_0078_AT2001_5250_0019_AT2001_5250AT2001_33A3DF1B80"}
{attribute addProperty CRC "2918768554"}
{attribute addProperty Size "80"}
{attribute addProperty Name "A_0066(AT2026-0250-0020) (AT2026-0250)"}
TYPE A_0066_AT2026_0250_0020_AT2026_0250_ADF8DFAA EXTENDS AT2026_2EA6C9BF :
STRUCT
	{attribute addProperty Name "A_0078(AT2001-5250-0019) (AT2001-5250)"}
	{attribute addProperty PreviousPort "A_0066(AT2026-0250-0020) (AT2026-0250) : B"}
	A_0078_AT2001_5250_0019_AT2001_5250 : AT2001_33A3DF1B;
END_STRUCT
END_TYPE

// ---- DUTs/IO/Topology/A_0067_AT2026_0250_0022_AT2026_0250_BF728FE6.TcDUT
{attribute 'GeneratedUsingTerminal: AT2026-0250-0022'}
{attribute addProperty BoxType "AT2026-0250-0022"}
{attribute addProperty Id "A_0079_AT2002_5249_0018_AT2002_5249AT2002_33A3DF1B80"}
{attribute addProperty CRC "3211956198"}
{attribute addProperty Size "80"}
{attribute addProperty Name "A_0067(AT2026-0250-0022) (AT2026-0250)"}
TYPE A_0067_AT2026_0250_0022_AT2026_0250_BF728FE6 EXTENDS AT2026_2EA6C9BF :
STRUCT
	{attribute addProperty Name "A_0079(AT2002-5249-0018) (AT2002-5249)"}
	{attribute addProperty PreviousPort "A_0067(AT2026-0250-0022) (AT2026-0250) : B"}
	A_0079_AT2002_5249_0018_AT2002_5249 : AT2002_33A3DF1B;
END_STRUCT
END_TYPE

// ---- DUTs/IO/Topology/A_0068_AT2026_0250_0024_AT2026_0250_71C01165.TcDUT
{attribute 'GeneratedUsingTerminal: AT2026-0250-0024'}
{attribute addProperty BoxType "AT2026-0250-0024"}
{attribute addProperty Id "A_0080_AT2002_5249_0019_AT2002_5249AT2002_33A3DF1B80"}
{attribute addProperty CRC "1908412773"}
{attribute addProperty Size "80"}
{attribute addProperty Name "A_0068(AT2026-0250-0024) (AT2026-0250)"}
TYPE A_0068_AT2026_0250_0024_AT2026_0250_71C01165 EXTENDS AT2026_2EA6C9BF :
STRUCT
	{attribute addProperty Name "A_0080(AT2002-5249-0019) (AT2002-5249)"}
	{attribute addProperty PreviousPort "A_0068(AT2026-0250-0024) (AT2026-0250) : B"}
	A_0080_AT2002_5249_0019_AT2002_5249 : AT2002_33A3DF1B;
END_STRUCT
END_TYPE

// ---- DUTs/IO/Topology/A_0069_AT2050_0501_0019_AT2050_0501_10255FA6.TcDUT
{attribute 'GeneratedUsingTerminal: AT2050-0501-0019'}
{attribute addProperty BoxType "AT2050-0501-0019"}
{attribute addProperty Id "A_0081_AT2002_5250_0018_AT2002_5250AT2002_33A3DF1B80"}
{attribute addProperty CRC "270884774"}
{attribute addProperty Size "80"}
{attribute addProperty Name "A_0069(AT2050-0501-0019) (AT2050-0501)"}
TYPE A_0069_AT2050_0501_0019_AT2050_0501_10255FA6 EXTENDS AT2050_2EA6C9BF :
STRUCT
	{attribute addProperty Name "A_0081(AT2002-5250-0018) (AT2002-5250)"}
	{attribute addProperty PreviousPort "A_0069(AT2050-0501-0019) (AT2050-0501) : B"}
	A_0081_AT2002_5250_0018_AT2002_5250 : AT2002_33A3DF1B;
END_STRUCT
END_TYPE

// ---- DUTs/IO/Topology/A_0070_AT2050_0501_0022_AT2050_0501_E445CD40.TcDUT
{attribute 'GeneratedUsingTerminal: AT2050-0501-0022'}
{attribute addProperty BoxType "AT2050-0501-0022"}
{attribute addProperty Id "A_0082_AT2002_5250_0019_AT2002_5250AT2002_33A3DF1B80"}
{attribute addProperty CRC "3829779776"}
{attribute addProperty Size "80"}
{attribute addProperty Name "A_0070(AT2050-0501-0022) (AT2050-0501)"}
TYPE A_0070_AT2050_0501_0022_AT2050_0501_E445CD40 EXTENDS AT2050_2EA6C9BF :
STRUCT
	{attribute addProperty Name "A_0082(AT2002-5250-0019) (AT2002-5250)"}
	{attribute addProperty PreviousPort "A_0070(AT2050-0501-0022) (AT2050-0501) : B"}
	A_0082_AT2002_5250_0019_AT2002_5250 : AT2002_33A3DF1B;
END_STRUCT
END_TYPE

// ---- DUTs/IO/Topology/A_0071_AT2050_0501_0023_AT2050_0501_A5CC9684.TcDUT
{attribute 'GeneratedUsingTerminal: AT2050-0501-0023'}
{attribute addProperty BoxType "AT2050-0501-0023"}
{attribute addProperty Id "A_0083_AT2050_5500_0016_AT2050_5500AT2050_33A3DF1B80"}
{attribute addProperty CRC "2781648516"}
{attribute addProperty Size "80"}
{attribute addProperty Name "A_0071(AT2050-0501-0023) (AT2050-0501)"}
TYPE A_0071_AT2050_0501_0023_AT2050_0501_A5CC9684 EXTENDS AT2050_2EA6C9BF :
STRUCT
	{attribute addProperty Name "A_0083(AT2050-5500-0016) (AT2050-5500)"}
	{attribute addProperty PreviousPort "A_0071(AT2050-0501-0023) (AT2050-0501) : B"}
	A_0083_AT2050_5500_0016_AT2050_5500 : AT2050_33A3DF1B;
END_STRUCT
END_TYPE

// ---- DUTs/IO/Topology/A_0072_AT2050_0501_0024_AT2050_0501_05E6D620.TcDUT
{attribute 'GeneratedUsingTerminal: AT2050-0501-0024'}
{attribute addProperty BoxType "AT2050-0501-0024"}
{attribute addProperty Id "A_0084_AT2050_5500_0017_AT2050_5500AT2050_33A3DF1B80"}
{attribute addProperty CRC "99014176"}
{attribute addProperty Size "80"}
{attribute addProperty Name "A_0072(AT2050-0501-0024) (AT2050-0501)"}
TYPE A_0072_AT2050_0501_0024_AT2050_0501_05E6D620 EXTENDS AT2050_2EA6C9BF :
STRUCT
	{attribute addProperty Name "A_0084(AT2050-5500-0017) (AT2050-5500)"}
	{attribute addProperty PreviousPort "A_0072(AT2050-0501-0024) (AT2050-0501) : B"}
	A_0084_AT2050_5500_0017_AT2050_5500 : AT2050_33A3DF1B;
END_STRUCT
END_TYPE

// ---- DUTs/IO/Topology/Beckhoff_AT2xxxEK1122_43DD63D7.TcDUT
{attribute 'GeneratedUsingTerminal: EK1122-0000-0018'}
{attribute addProperty BoxType "EK1122-0000-0018"}
{attribute addProperty Id "A_0060_AT2020_0250_0019_AT2020_0250A_0060_AT2020_0250_0019_AT2020_0250_29EE827680Beckhoff_AT2xxxsub_EK1100EK1100_1FC0878B2A_0001_AT2000_0233_0022AT2000_1809CD2F80A_0002_AT2000_0233_0023AT2000_1809CD2F80A_0003_AT2000_0233_0024AT2000_1809CD2F80A_0004_AT2000_0250_0016AT2000_2EA6C9BF84A_0005_AT2000_0250_0017AT2000_2EA6C9BF84A_0006_AT2000_0250_0018AT2000_2EA6C9BF84A_0007_AT2000_0250_0019AT2000_2EA6C9BF84A_0008_AT2000_0250_0020AT2000_2EA6C9BF84A_0009_AT2000_0250_0021AT2000_2EA6C9BF84A_0010_AT2000_0250_0022AT2000_2EA6C9BF84A_0011_AT2000_0250_0023AT2000_2EA6C9BF84A_0012_AT2001_0250_0016AT2001_2EA6C9BF84A_0013_AT2001_0250_0017AT2001_2EA6C9BF84A_0014_AT2001_0250_0018AT2001_2EA6C9BF84A_0015_AT2001_0250_0019AT2001_2EA6C9BF84A_0016_AT2001_0250_0020AT2001_2EA6C9BF84A_0017_AT2001_0250_0022AT2001_2EA6C9BF84A_0018_AT2001_0250_0023AT2001_2EA6C9BF84A_0019_AT2001_0250_0024AT2001_2EA6C9BF84A_0020_AT2002_0249_0021AT2002_2EA6C9BF84A_0021_AT2002_0249_0022AT2002_2EA6C9BF84A_0022_AT2002_0249_0023AT2002_2EA6C9BF84A_0023_AT2002_0250_0022AT2002_2EA6C9BF84A_0024_AT2002_0250_0023AT2002_2EA6C9BF84A_0025_AT2002_0250_0024AT2002_2EA6C9BF84A_0026_AT2020_0250_0018AT2020_2EA6C9BF84A_0027_AT2020_0250_0021AT2020_2EA6C9BF84A_0028_AT2021_0250_0018AT2021_2EA6C9BF84A_0029_AT2021_0250_0020AT2021_2EA6C9BF84A_0030_AT2025_0250_0018AT2025_2EA6C9BF84A_0031_AT2026_0250_0021AT2026_2EA6C9BF84A_0032_AT2026_0250_0023AT2026_2EA6C9BF84A_0033_AT2040_0250_0018AT2040_2EA6C9BF84A_0034_AT2040_0250_0019AT2040_2EA6C9BF84A_0035_AT2040_0250_0020AT2040_2EA6C9BF84A_0036_AT2040_0250_0021A_0036_AT2040_0250_0021_0B822AE480A_0037_AT2040_0250_0022A_0037_AT2040_0250_0022_033DCEC480A_0038_AT2040_0250_0023A_0038_AT2040_0250_0023_C339CA0C80A_0039_AT2040_0250_0024A_0039_AT2040_0250_0024_375958EA80A_0040_AT2041_0250_0018A_0040_AT2041_0250_0018_536500F280A_0041_AT2041_0250_0019A_0041_AT2041_0250_0019_F34F405680A_0042_AT2041_0250_0020A_0042_AT2041_0250_0020_5E65A51E80A_0043_AT2041_0250_0021A_0043_AT2041_0250_0021_AA0537F880A_0044_AT2041_0250_0022A_0044_AT2041_0250_0022_5A9A39BA80A_0045_AT2041_0250_0023A_0045_AT2041_0250_0023_51C662AC80A_0046_AT2042_0250_0024A_0046_AT2042_0250_0024_1B20CF3180A_0047_AT2050_0500_0016A_0047_AT2050_0500_0016_139F2B1180A_0048_AT2050_0500_0017A_0048_AT2050_0500_0017_3F977F4780A_0049_AT2050_0500_0018A_0049_AT2050_0500_0018_CBE655A880A_0050_AT2050_0500_0019A_0050_AT2050_0500_0019_15A3AE6F80A_0051_AT2050_0500_0020A_0051_AT2050_0500_0020_9B531B4E80A_0052_AT2050_0500_0021A_0052_AT2050_0500_0021_4516E08980A_0053_AT2050_0500_0022A_0053_AT2050_0500_0022_433BDDFE80A_0054_AT2050_0500_0023A_0054_AT2050_0500_0023_B2F2DF5580A_0055_AT2050_0500_0024A_0055_AT2050_0500_0024_8D42A08D80A_0056_AT2050_0501_0017A_0056_AT2050_0501_0017_A14AF4DB80A_0057_AT2050_0501_0020A_0057_AT2050_0501_0020_A9F510FB80A_0058_AT2050_0501_0021A_0058_AT2050_0501_0021_DD8E109080A_0061_AT2020_0250_0023_AT2020_0250A_0061_AT2020_0250_0023_AT2020_0250_2D9AB3DC80A_0062_AT2025_0250_0020_AT2025_0250A_0062_AT2025_0250_0020_AT2025_0250_8DB0F37880A_0063_AT2025_0250_0022_AT2025_0250A_0063_AT2025_0250_0022_AT2025_0250_E88F66A280A_0064_AT2025_0250_0023_AT2025_0250A_0064_AT2025_0250_0023_AT2025_0250_894F6FDC80A_0065_AT2026_0250_0019_AT2026_0250A_0065_AT2026_0250_0019_AT2026_0250_A5473B8A80A_0066_AT2026_0250_0020_AT2026_0250A_0066_AT2026_0250_0020_AT2026_0250_ADF8DFAA80A_0067_AT2026_0250_0022_AT2026_0250A_0067_AT2026_0250_0022_AT2026_0250_BF728FE680A_0068_AT2026_0250_0024_AT2026_0250A_0068_AT2026_0250_0024_AT2026_0250_71C0116580A_0069_AT2050_0501_0019_AT2050_0501A_0069_AT2050_0501_0019_AT2050_0501_10255FA680A_0070_AT2050_0501_0022_AT2050_0501A_0070_AT2050_0501_0022_AT2050_0501_E445CD4080A_0071_AT2050_0501_0023_AT2050_0501A_0071_AT2050_0501_0023_AT2050_0501_A5CC968480A_0072_AT2050_0501_0024_AT2050_0501A_0072_AT2050_0501_0024_AT2050_0501_05E6D62080"}
{attribute addProperty CRC "1138582487"}
{attribute addProperty Size "5810"}
{attribute addProperty Name "Beckhoff AT2xxxEK1122"}
TYPE Beckhoff_AT2xxxEK1122_43DD63D7 EXTENDS EK1122_1FC0878B :
STRUCT
	{attribute addProperty Name "A_0060(AT2020-0250-0019) (AT2020-0250)"}
	{attribute addProperty PreviousPort "Beckhoff AT2xxxEK1122 : D"}
	A_0060_AT2020_0250_0019_AT2020_0250 : A_0060_AT2020_0250_0019_AT2020_0250_29EE8276;
	{attribute addProperty Name "Beckhoff AT2xxxsub EK1100"}
	{attribute addProperty PreviousPort "A_0060(AT2020-0250-0019) (AT2020-0250) : C"}
	Beckhoff_AT2xxxsub_EK1100 : EK1100_1FC0878B;
	{attribute addProperty Name "A_0001(AT2000-0233-0022)"}
	{attribute addProperty PreviousPort "Beckhoff AT2xxxsub EK1100 : C"}
	A_0001_AT2000_0233_0022 : AT2000_1809CD2F;
	{attribute addProperty Name "A_0002(AT2000-0233-0023)"}
	{attribute addProperty PreviousPort "A_0001(AT2000-0233-0022) : C"}
	A_0002_AT2000_0233_0023 : AT2000_1809CD2F;
	{attribute addProperty Name "A_0003(AT2000-0233-0024)"}
	{attribute addProperty PreviousPort "A_0002(AT2000-0233-0023) : C"}
	A_0003_AT2000_0233_0024 : AT2000_1809CD2F;
	{attribute addProperty Name "A_0004(AT2000-0250-0016)"}
	{attribute addProperty PreviousPort "A_0003(AT2000-0233-0024) : C"}
	A_0004_AT2000_0250_0016 : AT2000_2EA6C9BF;
	{attribute addProperty Name "A_0005(AT2000-0250-0017)"}
	{attribute addProperty PreviousPort "A_0004(AT2000-0250-0016) : C"}
	A_0005_AT2000_0250_0017 : AT2000_2EA6C9BF;
	{attribute addProperty Name "A_0006(AT2000-0250-0018)"}
	{attribute addProperty PreviousPort "A_0005(AT2000-0250-0017) : C"}
	A_0006_AT2000_0250_0018 : AT2000_2EA6C9BF;
	{attribute addProperty Name "A_0007(AT2000-0250-0019)"}
	{attribute addProperty PreviousPort "A_0006(AT2000-0250-0018) : C"}
	A_0007_AT2000_0250_0019 : AT2000_2EA6C9BF;
	{attribute addProperty Name "A_0008(AT2000-0250-0020)"}
	{attribute addProperty PreviousPort "A_0007(AT2000-0250-0019) : C"}
	A_0008_AT2000_0250_0020 : AT2000_2EA6C9BF;
	{attribute addProperty Name "A_0009(AT2000-0250-0021)"}
	{attribute addProperty PreviousPort "A_0008(AT2000-0250-0020) : C"}
	A_0009_AT2000_0250_0021 : AT2000_2EA6C9BF;
	{attribute addProperty Name "A_0010(AT2000-0250-0022)"}
	{attribute addProperty PreviousPort "A_0009(AT2000-0250-0021) : C"}
	A_0010_AT2000_0250_0022 : AT2000_2EA6C9BF;
	{attribute addProperty Name "A_0011(AT2000-0250-0023)"}
	{attribute addProperty PreviousPort "A_0010(AT2000-0250-0022) : C"}
	A_0011_AT2000_0250_0023 : AT2000_2EA6C9BF;
	{attribute addProperty Name "A_0012(AT2001-0250-0016)"}
	{attribute addProperty PreviousPort "A_0011(AT2000-0250-0023) : C"}
	A_0012_AT2001_0250_0016 : AT2001_2EA6C9BF;
	{attribute addProperty Name "A_0013(AT2001-0250-0017)"}
	{attribute addProperty PreviousPort "A_0012(AT2001-0250-0016) : C"}
	A_0013_AT2001_0250_0017 : AT2001_2EA6C9BF;
	{attribute addProperty Name "A_0014(AT2001-0250-0018)"}
	{attribute addProperty PreviousPort "A_0013(AT2001-0250-0017) : C"}
	A_0014_AT2001_0250_0018 : AT2001_2EA6C9BF;
	{attribute addProperty Name "A_0015(AT2001-0250-0019)"}
	{attribute addProperty PreviousPort "A_0014(AT2001-0250-0018) : C"}
	A_0015_AT2001_0250_0019 : AT2001_2EA6C9BF;
	{attribute addProperty Name "A_0016(AT2001-0250-0020)"}
	{attribute addProperty PreviousPort "A_0015(AT2001-0250-0019) : C"}
	A_0016_AT2001_0250_0020 : AT2001_2EA6C9BF;
	{attribute addProperty Name "A_0017(AT2001-0250-0022)"}
	{attribute addProperty PreviousPort "A_0016(AT2001-0250-0020) : C"}
	A_0017_AT2001_0250_0022 : AT2001_2EA6C9BF;
	{attribute addProperty Name "A_0018(AT2001-0250-0023)"}
	{attribute addProperty PreviousPort "A_0017(AT2001-0250-0022) : C"}
	A_0018_AT2001_0250_0023 : AT2001_2EA6C9BF;
	{attribute addProperty Name "A_0019(AT2001-0250-0024)"}
	{attribute addProperty PreviousPort "A_0018(AT2001-0250-0023) : C"}
	A_0019_AT2001_0250_0024 : AT2001_2EA6C9BF;
	{attribute addProperty Name "A_0020(AT2002-0249-0021)"}
	{attribute addProperty PreviousPort "A_0019(AT2001-0250-0024) : C"}
	A_0020_AT2002_0249_0021 : AT2002_2EA6C9BF;
	{attribute addProperty Name "A_0021(AT2002-0249-0022)"}
	{attribute addProperty PreviousPort "A_0020(AT2002-0249-0021) : C"}
	A_0021_AT2002_0249_0022 : AT2002_2EA6C9BF;
	{attribute addProperty Name "A_0022(AT2002-0249-0023)"}
	{attribute addProperty PreviousPort "A_0021(AT2002-0249-0022) : C"}
	A_0022_AT2002_0249_0023 : AT2002_2EA6C9BF;
	{attribute addProperty Name "A_0023(AT2002-0250-0022)"}
	{attribute addProperty PreviousPort "A_0022(AT2002-0249-0023) : C"}
	A_0023_AT2002_0250_0022 : AT2002_2EA6C9BF;
	{attribute addProperty Name "A_0024(AT2002-0250-0023)"}
	{attribute addProperty PreviousPort "A_0023(AT2002-0250-0022) : C"}
	A_0024_AT2002_0250_0023 : AT2002_2EA6C9BF;
	{attribute addProperty Name "A_0025(AT2002-0250-0024)"}
	{attribute addProperty PreviousPort "A_0024(AT2002-0250-0023) : C"}
	A_0025_AT2002_0250_0024 : AT2002_2EA6C9BF;
	{attribute addProperty Name "A_0026(AT2020-0250-0018)"}
	{attribute addProperty PreviousPort "A_0025(AT2002-0250-0024) : C"}
	A_0026_AT2020_0250_0018 : AT2020_2EA6C9BF;
	{attribute addProperty Name "A_0027(AT2020-0250-0021)"}
	{attribute addProperty PreviousPort "A_0026(AT2020-0250-0018) : C"}
	A_0027_AT2020_0250_0021 : AT2020_2EA6C9BF;
	{attribute addProperty Name "A_0028(AT2021-0250-0018)"}
	{attribute addProperty PreviousPort "A_0027(AT2020-0250-0021) : C"}
	A_0028_AT2021_0250_0018 : AT2021_2EA6C9BF;
	{attribute addProperty Name "A_0029(AT2021-0250-0020)"}
	{attribute addProperty PreviousPort "A_0028(AT2021-0250-0018) : C"}
	A_0029_AT2021_0250_0020 : AT2021_2EA6C9BF;
	{attribute addProperty Name "A_0030(AT2025-0250-0018)"}
	{attribute addProperty PreviousPort "A_0029(AT2021-0250-0020) : C"}
	A_0030_AT2025_0250_0018 : AT2025_2EA6C9BF;
	{attribute addProperty Name "A_0031(AT2026-0250-0021)"}
	{attribute addProperty PreviousPort "A_0030(AT2025-0250-0018) : C"}
	A_0031_AT2026_0250_0021 : AT2026_2EA6C9BF;
	{attribute addProperty Name "A_0032(AT2026-0250-0023)"}
	{attribute addProperty PreviousPort "A_0031(AT2026-0250-0021) : C"}
	A_0032_AT2026_0250_0023 : AT2026_2EA6C9BF;
	{attribute addProperty Name "A_0033(AT2040-0250-0018)"}
	{attribute addProperty PreviousPort "A_0032(AT2026-0250-0023) : C"}
	A_0033_AT2040_0250_0018 : AT2040_2EA6C9BF;
	{attribute addProperty Name "A_0034(AT2040-0250-0019)"}
	{attribute addProperty PreviousPort "A_0033(AT2040-0250-0018) : C"}
	A_0034_AT2040_0250_0019 : AT2040_2EA6C9BF;
	{attribute addProperty Name "A_0035(AT2040-0250-0020)"}
	{attribute addProperty PreviousPort "A_0034(AT2040-0250-0019) : C"}
	A_0035_AT2040_0250_0020 : AT2040_2EA6C9BF;
	{attribute addProperty Name "A_0036(AT2040-0250-0021)"}
	{attribute addProperty PreviousPort "A_0035(AT2040-0250-0020) : C"}
	A_0036_AT2040_0250_0021 : A_0036_AT2040_0250_0021_0B822AE4;
	{attribute addProperty Name "A_0037(AT2040-0250-0022)"}
	{attribute addProperty PreviousPort "A_0036(AT2040-0250-0021) : C"}
	A_0037_AT2040_0250_0022 : A_0037_AT2040_0250_0022_033DCEC4;
	{attribute addProperty Name "A_0038(AT2040-0250-0023)"}
	{attribute addProperty PreviousPort "A_0037(AT2040-0250-0022) : C"}
	A_0038_AT2040_0250_0023 : A_0038_AT2040_0250_0023_C339CA0C;
	{attribute addProperty Name "A_0039(AT2040-0250-0024)"}
	{attribute addProperty PreviousPort "A_0038(AT2040-0250-0023) : C"}
	A_0039_AT2040_0250_0024 : A_0039_AT2040_0250_0024_375958EA;
	{attribute addProperty Name "A_0040(AT2041-0250-0018)"}
	{attribute addProperty PreviousPort "A_0039(AT2040-0250-0024) : C"}
	A_0040_AT2041_0250_0018 : A_0040_AT2041_0250_0018_536500F2;
	{attribute addProperty Name "A_0041(AT2041-0250-0019)"}
	{attribute addProperty PreviousPort "A_0040(AT2041-0250-0018) : C"}
	A_0041_AT2041_0250_0019 : A_0041_AT2041_0250_0019_F34F4056;
	{attribute addProperty Name "A_0042(AT2041-0250-0020)"}
	{attribute addProperty PreviousPort "A_0041(AT2041-0250-0019) : C"}
	A_0042_AT2041_0250_0020 : A_0042_AT2041_0250_0020_5E65A51E;
	{attribute addProperty Name "A_0043(AT2041-0250-0021)"}
	{attribute addProperty PreviousPort "A_0042(AT2041-0250-0020) : C"}
	A_0043_AT2041_0250_0021 : A_0043_AT2041_0250_0021_AA0537F8;
	{attribute addProperty Name "A_0044(AT2041-0250-0022)"}
	{attribute addProperty PreviousPort "A_0043(AT2041-0250-0021) : C"}
	A_0044_AT2041_0250_0022 : A_0044_AT2041_0250_0022_5A9A39BA;
	{attribute addProperty Name "A_0045(AT2041-0250-0023)"}
	{attribute addProperty PreviousPort "A_0044(AT2041-0250-0022) : C"}
	A_0045_AT2041_0250_0023 : A_0045_AT2041_0250_0023_51C662AC;
	{attribute addProperty Name "A_0046(AT2042-0250-0024)"}
	{attribute addProperty PreviousPort "A_0045(AT2041-0250-0023) : C"}
	A_0046_AT2042_0250_0024 : A_0046_AT2042_0250_0024_1B20CF31;
	{attribute addProperty Name "A_0047(AT2050-0500-0016)"}
	{attribute addProperty PreviousPort "A_0046(AT2042-0250-0024) : C"}
	A_0047_AT2050_0500_0016 : A_0047_AT2050_0500_0016_139F2B11;
	{attribute addProperty Name "A_0048(AT2050-0500-0017)"}
	{attribute addProperty PreviousPort "A_0047(AT2050-0500-0016) : C"}
	A_0048_AT2050_0500_0017 : A_0048_AT2050_0500_0017_3F977F47;
	{attribute addProperty Name "A_0049(AT2050-0500-0018)"}
	{attribute addProperty PreviousPort "A_0048(AT2050-0500-0017) : C"}
	A_0049_AT2050_0500_0018 : A_0049_AT2050_0500_0018_CBE655A8;
	{attribute addProperty Name "A_0050(AT2050-0500-0019)"}
	{attribute addProperty PreviousPort "A_0049(AT2050-0500-0018) : C"}
	A_0050_AT2050_0500_0019 : A_0050_AT2050_0500_0019_15A3AE6F;
	{attribute addProperty Name "A_0051(AT2050-0500-0020)"}
	{attribute addProperty PreviousPort "A_0050(AT2050-0500-0019) : C"}
	A_0051_AT2050_0500_0020 : A_0051_AT2050_0500_0020_9B531B4E;
	{attribute addProperty Name "A_0052(AT2050-0500-0021)"}
	{attribute addProperty PreviousPort "A_0051(AT2050-0500-0020) : C"}
	A_0052_AT2050_0500_0021 : A_0052_AT2050_0500_0021_4516E089;
	{attribute addProperty Name "A_0053(AT2050-0500-0022)"}
	{attribute addProperty PreviousPort "A_0052(AT2050-0500-0021) : C"}
	A_0053_AT2050_0500_0022 : A_0053_AT2050_0500_0022_433BDDFE;
	{attribute addProperty Name "A_0054(AT2050-0500-0023)"}
	{attribute addProperty PreviousPort "A_0053(AT2050-0500-0022) : C"}
	A_0054_AT2050_0500_0023 : A_0054_AT2050_0500_0023_B2F2DF55;
	{attribute addProperty Name "A_0055(AT2050-0500-0024)"}
	{attribute addProperty PreviousPort "A_0054(AT2050-0500-0023) : C"}
	A_0055_AT2050_0500_0024 : A_0055_AT2050_0500_0024_8D42A08D;
	{attribute addProperty Name "A_0056(AT2050-0501-0017)"}
	{attribute addProperty PreviousPort "A_0055(AT2050-0500-0024) : C"}
	A_0056_AT2050_0501_0017 : A_0056_AT2050_0501_0017_A14AF4DB;
	{attribute addProperty Name "A_0057(AT2050-0501-0020)"}
	{attribute addProperty PreviousPort "A_0056(AT2050-0501-0017) : C"}
	A_0057_AT2050_0501_0020 : A_0057_AT2050_0501_0020_A9F510FB;
	{attribute addProperty Name "A_0058(AT2050-0501-0021)"}
	{attribute addProperty PreviousPort "A_0057(AT2050-0501-0020) : C"}
	A_0058_AT2050_0501_0021 : A_0058_AT2050_0501_0021_DD8E1090;
	{attribute addProperty Name "A_0061(AT2020-0250-0023) (AT2020-0250)"}
	{attribute addProperty PreviousPort "Beckhoff AT2xxxEK1122 : B"}
	A_0061_AT2020_0250_0023_AT2020_0250 : A_0061_AT2020_0250_0023_AT2020_0250_2D9AB3DC;
	{attribute addProperty Name "A_0062(AT2025-0250-0020) (AT2025-0250)"}
	{attribute addProperty PreviousPort "A_0061(AT2020-0250-0023) (AT2020-0250) : C"}
	A_0062_AT2025_0250_0020_AT2025_0250 : A_0062_AT2025_0250_0020_AT2025_0250_8DB0F378;
	{attribute addProperty Name "A_0063(AT2025-0250-0022) (AT2025-0250)"}
	{attribute addProperty PreviousPort "A_0062(AT2025-0250-0020) (AT2025-0250) : C"}
	A_0063_AT2025_0250_0022_AT2025_0250 : A_0063_AT2025_0250_0022_AT2025_0250_E88F66A2;
	{attribute addProperty Name "A_0064(AT2025-0250-0023) (AT2025-0250)"}
	{attribute addProperty PreviousPort "A_0063(AT2025-0250-0022) (AT2025-0250) : C"}
	A_0064_AT2025_0250_0023_AT2025_0250 : A_0064_AT2025_0250_0023_AT2025_0250_894F6FDC;
	{attribute addProperty Name "A_0065(AT2026-0250-0019) (AT2026-0250)"}
	{attribute addProperty PreviousPort "A_0064(AT2025-0250-0023) (AT2025-0250) : C"}
	A_0065_AT2026_0250_0019_AT2026_0250 : A_0065_AT2026_0250_0019_AT2026_0250_A5473B8A;
	{attribute addProperty Name "A_0066(AT2026-0250-0020) (AT2026-0250)"}
	{attribute addProperty PreviousPort "A_0065(AT2026-0250-0019) (AT2026-0250) : C"}
	A_0066_AT2026_0250_0020_AT2026_0250 : A_0066_AT2026_0250_0020_AT2026_0250_ADF8DFAA;
	{attribute addProperty Name "A_0067(AT2026-0250-0022) (AT2026-0250)"}
	{attribute addProperty PreviousPort "A_0066(AT2026-0250-0020) (AT2026-0250) : C"}
	A_0067_AT2026_0250_0022_AT2026_0250 : A_0067_AT2026_0250_0022_AT2026_0250_BF728FE6;
	{attribute addProperty Name "A_0068(AT2026-0250-0024) (AT2026-0250)"}
	{attribute addProperty PreviousPort "A_0067(AT2026-0250-0022) (AT2026-0250) : C"}
	A_0068_AT2026_0250_0024_AT2026_0250 : A_0068_AT2026_0250_0024_AT2026_0250_71C01165;
	{attribute addProperty Name "A_0069(AT2050-0501-0019) (AT2050-0501)"}
	{attribute addProperty PreviousPort "A_0068(AT2026-0250-0024) (AT2026-0250) : C"}
	A_0069_AT2050_0501_0019_AT2050_0501 : A_0069_AT2050_0501_0019_AT2050_0501_10255FA6;
	{attribute addProperty Name "A_0070(AT2050-0501-0022) (AT2050-0501)"}
	{attribute addProperty PreviousPort "A_0069(AT2050-0501-0019) (AT2050-0501) : C"}
	A_0070_AT2050_0501_0022_AT2050_0501 : A_0070_AT2050_0501_0022_AT2050_0501_E445CD40;
	{attribute addProperty Name "A_0071(AT2050-0501-0023) (AT2050-0501)"}
	{attribute addProperty PreviousPort "A_0070(AT2050-0501-0022) (AT2050-0501) : C"}
	A_0071_AT2050_0501_0023_AT2050_0501 : A_0071_AT2050_0501_0023_AT2050_0501_A5CC9684;
	{attribute addProperty Name "A_0072(AT2050-0501-0024) (AT2050-0501)"}
	{attribute addProperty PreviousPort "A_0071(AT2050-0501-0023) (AT2050-0501) : C"}
	A_0072_AT2050_0501_0024_AT2050_0501 : A_0072_AT2050_0501_0024_AT2050_0501_05E6D620;
END_STRUCT
END_TYPE

// ---- DUTs/IO/Topology/Beckhoff_AT1xxx_27B72169.TcDUT
{attribute 'GeneratedUsingTerminal: EK1100-0000-0018'}
{attribute addProperty BoxType "EK1100-0000-0018"}
{attribute addProperty Id "Beckhoff_AT2xxxEK1122Beckhoff_AT2xxxEK1122_43DD63D75810A_0059_AT2000_5250_0018AT2000_33A3DF1B80"}
{attribute addProperty CRC "666313065"}
{attribute addProperty Size "5890"}
{attribute addProperty Name "Beckhoff AT1xxx"}
TYPE Beckhoff_AT1xxx_27B72169 EXTENDS EK1100_1FC0878B :
STRUCT
	{attribute addProperty Name "Beckhoff AT2xxxEK1122"}
	{attribute addProperty PreviousPort "Beckhoff AT1xxx : B"}
	Beckhoff_AT2xxxEK1122 : Beckhoff_AT2xxxEK1122_43DD63D7;
	{attribute addProperty Name "A_0059(AT2000-5250-0018)"}
	{attribute addProperty PreviousPort "Beckhoff AT2xxxEK1122 : C"}
	A_0059_AT2000_5250_0018 : AT2000_33A3DF1B;
END_STRUCT
END_TYPE

// ---- DUTs/IO/Topology/A_0001_ATH2000_0250_0022_300D1FD0.TcDUT
{attribute 'GeneratedUsingTerminal: ATH2000-0250-0022'}
{attribute addProperty BoxType "ATH2000-0250-0022"}
{attribute addProperty Id "A_0014_ATH2050_5501_0022ATH2050_6EC099B714"}
{attribute addProperty CRC "806166480"}
{attribute addProperty Size "14"}
{attribute addProperty Name "A_0001(ATH2000-0250-0022)"}
TYPE A_0001_ATH2000_0250_0022_300D1FD0 EXTENDS ATH2000_2EA6C9BF :
STRUCT
	{attribute addProperty Name "A_0014(ATH2050-5501-0022)"}
	{attribute addProperty PreviousPort "A_0001(ATH2000-0250-0022) : B"}
	A_0014_ATH2050_5501_0022 : ATH2050_6EC099B7;
END_STRUCT
END_TYPE

// ---- DUTs/IO/Topology/A_0002_ATH2000_0250_0023_E62B11EA.TcDUT
{attribute 'GeneratedUsingTerminal: ATH2000-0250-0023'}
{attribute addProperty BoxType "ATH2000-0250-0023"}
{attribute addProperty Id "A_0015_ATH2040_5250_0022ATH2040_41437DDC14"}
{attribute addProperty CRC "3861582314"}
{attribute addProperty Size "14"}
{attribute addProperty Name "A_0002(ATH2000-0250-0023)"}
TYPE A_0002_ATH2000_0250_0023_E62B11EA EXTENDS ATH2000_2EA6C9BF :
STRUCT
	{attribute addProperty Name "A_0015(ATH2040-5250-0022)"}
	{attribute addProperty PreviousPort "A_0002(ATH2000-0250-0023) : B"}
	A_0015_ATH2040_5250_0022 : ATH2040_41437DDC;
END_STRUCT
END_TYPE

// ---- DUTs/IO/Topology/Beckhoff_ATH2xxxEK1122_61A38CAE.TcDUT
{attribute 'GeneratedUsingTerminal: EK1122-0000-0018'}
{attribute addProperty BoxType "EK1122-0000-0018"}
{attribute addProperty Id "Beckhoff_ATH2xxxsub_EK1100EK1100_1FC0878B2A_0001_ATH2000_0250_0022A_0001_ATH2000_0250_0022_300D1FD014A_0002_ATH2000_0250_0023A_0002_ATH2000_0250_0023_E62B11EA14A_0003_ATH2000_0250_0024ATH2000_2EA6C9BF84A_0004_ATH2040_0250_0022ATH2040_2EA6C9BF84A_0005_ATH2040_0250_0023ATH2040_2EA6C9BF84A_0006_ATH2040_0250_0024ATH2040_2EA6C9BF84A_0007_ATH2050_0500_0022ATH2050_2EA6C9BF84A_0008_ATH2050_0500_0023ATH2050_2EA6C9BF84A_0009_ATH2050_0500_0024ATH2050_2EA6C9BF84A_0010_ATH2050_0501_0022ATH2050_2EA6C9BF84A_0011_ATH2050_0501_0023ATH2050_2EA6C9BF84A_0012_ATH2050_0501_0024ATH2050_2EA6C9BF84"}
{attribute addProperty CRC "1638108334"}
{attribute addProperty Size "870"}
{attribute addProperty Name "Beckhoff ATH2xxxEK1122"}
TYPE Beckhoff_ATH2xxxEK1122_61A38CAE EXTENDS EK1122_1FC0878B :
STRUCT
	{attribute addProperty Name "Beckhoff ATH2xxxsub EK1100"}
	{attribute addProperty PreviousPort "Beckhoff ATH2xxxEK1122 : D"}
	Beckhoff_ATH2xxxsub_EK1100 : EK1100_1FC0878B;
	{attribute addProperty Name "A_0001(ATH2000-0250-0022)"}
	{attribute addProperty PreviousPort "Beckhoff ATH2xxxsub EK1100 : C"}
	A_0001_ATH2000_0250_0022 : A_0001_ATH2000_0250_0022_300D1FD0;
	{attribute addProperty Name "A_0002(ATH2000-0250-0023)"}
	{attribute addProperty PreviousPort "A_0001(ATH2000-0250-0022) : C"}
	A_0002_ATH2000_0250_0023 : A_0002_ATH2000_0250_0023_E62B11EA;
	{attribute addProperty Name "A_0003(ATH2000-0250-0024)"}
	{attribute addProperty PreviousPort "A_0002(ATH2000-0250-0023) : C"}
	A_0003_ATH2000_0250_0024 : ATH2000_2EA6C9BF;
	{attribute addProperty Name "A_0004(ATH2040-0250-0022)"}
	{attribute addProperty PreviousPort "A_0003(ATH2000-0250-0024) : C"}
	A_0004_ATH2040_0250_0022 : ATH2040_2EA6C9BF;
	{attribute addProperty Name "A_0005(ATH2040-0250-0023)"}
	{attribute addProperty PreviousPort "A_0004(ATH2040-0250-0022) : C"}
	A_0005_ATH2040_0250_0023 : ATH2040_2EA6C9BF;
	{attribute addProperty Name "A_0006(ATH2040-0250-0024)"}
	{attribute addProperty PreviousPort "A_0005(ATH2040-0250-0023) : C"}
	A_0006_ATH2040_0250_0024 : ATH2040_2EA6C9BF;
	{attribute addProperty Name "A_0007(ATH2050-0500-0022)"}
	{attribute addProperty PreviousPort "A_0006(ATH2040-0250-0024) : C"}
	A_0007_ATH2050_0500_0022 : ATH2050_2EA6C9BF;
	{attribute addProperty Name "A_0008(ATH2050-0500-0023)"}
	{attribute addProperty PreviousPort "A_0007(ATH2050-0500-0022) : C"}
	A_0008_ATH2050_0500_0023 : ATH2050_2EA6C9BF;
	{attribute addProperty Name "A_0009(ATH2050-0500-0024)"}
	{attribute addProperty PreviousPort "A_0008(ATH2050-0500-0023) : C"}
	A_0009_ATH2050_0500_0024 : ATH2050_2EA6C9BF;
	{attribute addProperty Name "A_0010(ATH2050-0501-0022)"}
	{attribute addProperty PreviousPort "A_0009(ATH2050-0500-0024) : C"}
	A_0010_ATH2050_0501_0022 : ATH2050_2EA6C9BF;
	{attribute addProperty Name "A_0011(ATH2050-0501-0023)"}
	{attribute addProperty PreviousPort "A_0010(ATH2050-0501-0022) : C"}
	A_0011_ATH2050_0501_0023 : ATH2050_2EA6C9BF;
	{attribute addProperty Name "A_0012(ATH2050-0501-0024)"}
	{attribute addProperty PreviousPort "A_0011(ATH2050-0501-0023) : C"}
	A_0012_ATH2050_0501_0024 : ATH2050_2EA6C9BF;
END_STRUCT
END_TYPE

// ---- DUTs/IO/Topology/Beckhoff_ATH2xxx_11442560.TcDUT
{attribute 'GeneratedUsingTerminal: EK1100-0000-0018'}
{attribute addProperty BoxType "EK1100-0000-0018"}
{attribute addProperty Id "Beckhoff_ATH2xxxEK1122Beckhoff_ATH2xxxEK1122_61A38CAE870A_0013_ATH2000_5250_0022ATH2000_D874080E14"}
{attribute addProperty CRC "289678688"}
{attribute addProperty Size "884"}
{attribute addProperty Name "Beckhoff ATH2xxx"}
TYPE Beckhoff_ATH2xxx_11442560 EXTENDS EK1100_1FC0878B :
STRUCT
	{attribute addProperty Name "Beckhoff ATH2xxxEK1122"}
	{attribute addProperty PreviousPort "Beckhoff ATH2xxx : B"}
	Beckhoff_ATH2xxxEK1122 : Beckhoff_ATH2xxxEK1122_61A38CAE;
	{attribute addProperty Name "A_0013(ATH2000-5250-0022)"}
	{attribute addProperty PreviousPort "Beckhoff ATH2xxxEK1122 : C"}
	A_0013_ATH2000_5250_0022 : ATH2000_D874080E;
END_STRUCT
END_TYPE

// ---- DUTs/IO/Topology/EtherCAT_Master_ATxxxx_981D2C79.TcDUT
{attribute 'GeneratedUsingTerminal: IODEVICETYPE_ETHERCATPROT'}
{attribute addProperty BoxType "IODEVICETYPE_ETHERCATPROT"}
{attribute addProperty Id "Beckhoff_AT1xxxBeckhoff_AT1xxx_27B721695890Beckhoff_ATH2xxxBeckhoff_ATH2xxx_11442560884SyncUnitsSyncUnits_99E584AF18InputsInputs_25A0042B160OutputsOutputs_2397A10E106InfoDataInfoData_E68C61CD28"}
{attribute addProperty CRC "2552048761"}
{attribute addProperty Size "7086"}
{attribute addProperty Name "EtherCAT Master ATxxxx"}
TYPE EtherCAT_Master_ATxxxx_981D2C79 EXTENDS EtcMasterBase_62654B43 :
STRUCT
	{attribute addProperty Name "Beckhoff AT1xxx"}
	{attribute addProperty PreviousPort "EtherCAT Master ATxxxx : Master"}
	Beckhoff_AT1xxx : Beckhoff_AT1xxx_27B72169;
	{attribute addProperty Name "Beckhoff ATH2xxx"}
	{attribute addProperty PreviousPort "Beckhoff AT1xxx : C"}
	Beckhoff_ATH2xxx : Beckhoff_ATH2xxx_11442560;
	{attribute addProperty Name "SyncUnits"}
	SyncUnits : SyncUnits_99E584AF;
	{attribute addProperty Name "Inputs"}
	Inputs : Inputs_25A0042B;
	{attribute addProperty Name "Outputs"}
	Outputs : Outputs_2397A10E;
	{attribute addProperty Name "InfoData"}
	InfoData : InfoData_E68C61CD;
END_STRUCT
END_TYPE

// ---- DUTs/IO/Base/EtcSlaveBase_82538BE2.TcDUT

TYPE EtcSlaveBase_82538BE2 :
STRUCT
END_STRUCT
END_TYPE

// ---- DUTs/IO/Base/EtcSlaveBase_82538BE2.TcDUT

TYPE EtcSlaveBase_82538BE2 :
STRUCT
END_STRUCT
END_TYPE

// ---- DUTs/IO/Base/EtcSlaveBase_82538BE2.TcDUT

TYPE EtcSlaveBase_82538BE2 :
STRUCT
END_STRUCT
END_TYPE

// ---- DUTs/IO/Base/EtcSlaveTerminalBase_947E5A46.TcDUT

{attribute clr[Container(Layout.Stack)]}
{attribute clr[Group(Layout.GroupBox)]}
{attribute addProperty PreviousPort "Unknown"}
TYPE EtcSlaveTerminalBase_947E5A46 EXTENDS EtcSlaveBase_82538BE2 :
STRUCT
END_STRUCT
END_TYPE

// ---- DUTs/IO/Base/EtcSlaveBoxBase_77A0E4A7.TcDUT

{attribute clr[Container(Layout.Stack)]}
{attribute clr[Group(Layout.GroupBox)]}
{attribute addProperty PreviousPort "Unknown"}
TYPE EtcSlaveBoxBase_77A0E4A7 EXTENDS EtcSlaveBase_82538BE2 :
STRUCT
END_STRUCT
END_TYPE

// ---- DUTs/IO/Base/EtcSlaveEndTerminalBase_866C7F0C.TcDUT

{attribute clr[Container(Layout.Stack)]}
{attribute clr[Group(Layout.GroupBox)]}
{attribute addProperty PreviousPort "Unknown"}
TYPE EtcSlaveEndTerminalBase_866C7F0C EXTENDS EtcSlaveBase_82538BE2 :
STRUCT
END_STRUCT
END_TYPE

// ---- DUTs/IO/Base/InputBase_8311D824.TcDUT

TYPE InputBase_8311D824 :
STRUCT
END_STRUCT
END_TYPE

// ---- DUTs/IO/Base/OutputBase_10CEE7DE.TcDUT

TYPE OutputBase_10CEE7DE :
STRUCT
END_STRUCT
END_TYPE

// ---- DUTs/IO/Base/EtcMasterBase_62654B43.TcDUT

TYPE EtcMasterBase_62654B43 :
STRUCT
END_STRUCT
END_TYPE

// ---- GVLs/GVL_iXlinker.TcGVL
{attribute 'qualified_only'}
VAR_GLOBAL
		EtherCAT_Master_ATxxxx : EtherCAT_Master_ATxxxx_981D2C79;
END_VAR

// ---- POUs/MAIN.TcPOU
PROGRAM MAIN
VAR
END_VAR

END_PROGRAM
